// TIA Portal V19 export
FUNCTION "LAF_SetPlcDateAndTime" : Void   // FC84, LAD
TITLE = LAF_SetPlcDateAndTime
AUTHOR : Siemens Digital Industries
FAMILY : LAF
VERSION : 1.2
// This set a new PLC time and date
// stored: Access Published, IsIECCheckEnabled true, SetENOAutomatically false
   VAR_INPUT
      setNewDateAndTime : Bool;   // Command to apply new time
      daylightSavingTime : Bool;   // TRUE = daylight saving time (first hour), FALSE = standard time (second hour)
   END_VAR
   VAR_IN_OUT
      newDateAndTime : Date_And_Time;   // New time that will be applied
   END_VAR
   VAR_TEMP
      tempLdtime : LDT;   // Temp LDT / Temporär LDT
      tempRetVal : Int;   // Temp return value Int / Temporärer Rückgabewert Int
   END_VAR
   VAR_TEMP   // added for the SCL form of the ladder/FBD networks
      _w1 : Bool;
   END_VAR
BEGIN

REGION Network 1: BLOCK INFO HEADER
   // SIEMENS AG / (c)Copyright 2024
   // ------------------------------------------------------------------------------
   // Title:            LAF_SetPlcDataAndTime
   // Comment/Function: This block sets a new local PLC time and date
   // Library/Family:   Library of Automation Framework
   // Author:                Siemens Digital Industry
   // Tested with:       S7-PLCSIM Advanced 6.0
   // Engineering:      TIA Portal V19
   // Restrictions:       ---
   // Requirements:   ---
   // ------------------------------------------------------------------------------
   // Change log table:
   // Version  | Date       | Expert in charge       | Changes applied
   // ---------|------------|------------------------|------------------------------
   // 01.01.00 | 21.06.2024 | SIMATIC Systems Support
   //                         First released version
   // 01.02.00 | 30.09.2024 | SIMATIC Systems Support
   //                         Block information properties updated
END_REGION

REGION Network 2: Set new time / SPS: Datum & Uhrzeit
   // Verwaltung von Datum und Uhrzeit der SPS. Konvertiergung dieser in verschiedene Formate und zuweisung auf den InOut Parameter
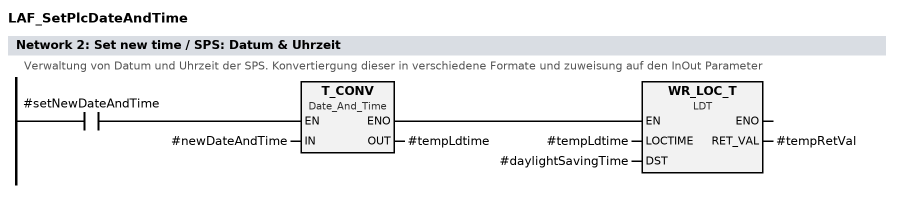
   RUNG wire#powerrail
      Contact( #setNewDateAndTime )
      { S7_Templates := "[src_type := Date_And_Time, dest_type := LDT]" } T_CONV(IN := #newDateAndTime, OUT => #tempLdtime)
      { S7_Templates := "loctime_type := LDT" } WR_LOC_T(LOCTIME := #tempLdtime, DST := #daylightSavingTime, Ret_Val => #tempRetVal)
   END_RUNG
   // the same network as SCL:
   T_CONV(EN := #setNewDateAndTime, IN := #newDateAndTime, OUT => #tempLdtime, ENO => #_w1);
   IF #_w1 THEN #tempRetVal := WR_LOC_T(LOCTIME := #tempLdtime, DST := #daylightSavingTime); END_IF;
END_REGION
END_FUNCTION
